Fanuc KAREL source: kc00030.KL

-- PROVISIONAL review KL for V1013-1; original PC SHA256 be8c040fa2e767ec41702ae2e66f1aacb2a161ec35e7ba27c13bbc5f172a7706
-- Incomplete behavior may be omitted. Consult companion uncertainty JSON. Do not deploy.
PROGRAM KC00030
%NOLOCKGROUP
BEGIN
  -- UNRESOLVED_PC offsets 5-17; opcodes 3F,75
  -- UNRESOLVED_PC offsets 22-94; opcodes 27,22,2A,22,22,22,22,22,22,22,22,22,22,31
  -- UNRESOLVED_PC offsets 99-103; opcodes 7F
END KC00030
